(* CoDeSys 2.3 export: ST_SE_CYLINDER_CFG.EXP *)

(* Data type *)
TYPE ST_SE_CYLINDER_CFG :
STRUCT
	Ease    : REAL; (*Usually 15% more than PMax*)
	Cycle   : REAL; (*Seconds*)
	TimeEase: REAL; (*Seconds*)
	TimeMax : REAL; (*Seconds*)
	HP      : BYTE; (*Num. Pumps*)
END_STRUCT
END_TYPE
